// TIA Portal V19 export
FUNCTION_BLOCK "TYPIC_C904_BF_SPI"   // FB44, FBD
TITLE = TYPIC_C904_BF_SPI: Schoonvloeistofpompinstallatie
{ S7_Optimized_Access := 'TRUE' }
AUTHOR : OCOTECH
FAMILY : Typical
NAME : C904.801
// Logisch Object Besturing: C904.801
// 
// 								Het doel van de BF SPI (schoonvloeistofpompinstallatie) is om de
// 								algemene sturing te voorzien van de schoonvloeistofpompinstallatie.
// 								De algemene sturing omvat het weergeven van de algemene toestand en
// 								het aano en afschakelen van pompen in functie van het vloeistofpeil
// 								en het actieve regime.
// stored: MemoryReserve 10, SetENOAutomatically false
   VAR_INPUT
      CFG_TST_UTYD { ExternalAccessible := 'False'; ExternalVisible := 'False'; ExternalWritable := 'False'} : Time;   // Time-out standverandering pompinstallatie (transitiestatus onbereikt)
      CFG_TST_OK_TYD { ExternalAccessible := 'False'; ExternalVisible := 'False'; ExternalWritable := 'False'} : Time;   // Stabilisatietijd voor de toestand OK (bereikt)
      CFG_NIV_H { ExternalAccessible := 'False'; ExternalVisible := 'False'; ExternalWritable := 'False'} : Real;   // Grenswaarde voor dreigende overloop (minder dan 30m3 bergruimte)
      CFG_NIV_HH { ExternalAccessible := 'False'; ExternalVisible := 'False'; ExternalWritable := 'False'} : Real;   // Grenswaarde voor overloop
      CFG_NIV_ITYD { ExternalAccessible := 'False'; ExternalVisible := 'False'; ExternalWritable := 'False'} : Time;   // Inschakelvertraging storingen grenswaarde
      CFG_NIV_HYS { ExternalAccessible := 'False'; ExternalVisible := 'False'; ExternalWritable := 'False'} : Real;   // Hysteresis storingen grenswaarde
      CFG_DEB_H { ExternalAccessible := 'False'; ExternalVisible := 'False'; ExternalWritable := 'False'} : Real;   // Grenswaarde minimaal debiet bij 1 aangeschakelde pomp
      CFG_DEB_HH { ExternalAccessible := 'False'; ExternalVisible := 'False'; ExternalWritable := 'False'} : Real;   // Grenswaarde minimaal debiet bij meerdere aangeschakelde pompen
      CFG_ITYD_DEB { ExternalAccessible := 'False'; ExternalVisible := 'False'; ExternalWritable := 'False'} : Time;   // Tijdsvertraging voor alarm afvoer verstopt (pomp aangeschakeld en minimaal debiet niet bereikt)
      STU_CMD_AUT { ExternalAccessible := 'False'; ExternalVisible := 'False'; ExternalWritable := 'False'} : USInt;   // Groepscommando: schakel in automatisch
      STU_CMD_WRE { ExternalAccessible := 'False'; ExternalVisible := 'False'; ExternalWritable := 'False'} : USInt;   // Sturing regime
      STU_ALG_LCK_SIG { ExternalAccessible := 'False'; ExternalVisible := 'False'; ExternalWritable := 'False'} : USInt;   // Onderdruk alarmen
   END_VAR
   VAR_OUTPUT
      VAR_PWR { ExternalAccessible := 'False'; ExternalVisible := 'False'; ExternalWritable := 'False'} : Real;   // Som actuele vermogens van alle pompen
      STU_PMP1 { ExternalAccessible := 'False'; ExternalVisible := 'False'; ExternalWritable := 'False'} : USInt;   // Sturing pomp
      STU_PMP2 { ExternalAccessible := 'False'; ExternalVisible := 'False'; ExternalWritable := 'False'} : USInt;   // Sturing pomp
      STU_PMP3 { ExternalAccessible := 'False'; ExternalVisible := 'False'; ExternalWritable := 'False'} : USInt;   // Sturing pomp
      STU_IF_SPI { ExternalAccessible := 'False'; ExternalVisible := 'False'; ExternalWritable := 'False'} : USInt;   // Gewenst regime (naar interne sturing)
   END_VAR
   VAR_IN_OUT
      VAR_IF_SPI : "C904_VAR_IF_SPI_TYPIC";   // Struct met variabelen ontvangen van de interne sturing van de pompinstallatie
      VAR_PMP : Array[*] of "C904_VAR_PMP_TYPIC";   // Array met alle pompen, met alle variabelen van de pomp
      VAR_NIV : "C904_VAR_NIV_TYPIC";   // Struct met alle variabelen ontvangen van de subfunctie niveaumeting
      VAR_DEB : "C904_VAR_DEB_TYPIC";   // Struct met alle variabelen ontvangen van de subfunctie debietmeting
   END_VAR
   VAR
      BED : Struct   // Bedieningen
         ALG : Struct   // Gewenste stand
            X : "UDT_BED_ALG";
            KNOP { S7_SetPoint := 'True'} : Array[0..3] of "UDT_BED_KNOP";
         END_STRUCT;
      END_STRUCT;
      BED_ALG { ExternalWritable := 'False'} : "TYPIC_HF_BED_ALG_KNOP";   // Gewenste stand
      SIG { ExternalWritable := 'False'} : Struct   // Signaleringen
         AA01 : Bool;   // Gewenste stand niet bereikt (transitiestatus = niet bereikt)
         AA02 : Bool;   // Schoonvloeistofpompinstallatie dreigt over te lopen
         AA03 : Bool;   // Overschrijding capaciteit schoonvloeistofpompinstallatie (overloop)
         AA04 : Bool;   // Afvoer verstopt en dreiging overloop van de schoonvloeistofpompinstallatie
         AA05 : Bool;   // Afvoer verstopt
         AB01 : Bool;   // Schoonvloeistofpompinstallatie niet beschikbaar
         AB02 : Bool;   // Schoonvloeistofpompinstallatie beperkt beschikbaar
         A001 : Bool;   // Beveiliging aangesproken
         A002 : Bool;   // Beveiliging No-Break aangesproken
         A003 : Bool;   // Overspanningsbeveiliging aangesproken
         A004 : Bool;   // Schuif ALSB uitgeschakeld
         A005 : Bool;   // Schuif ALSB in test
         A006 : Bool;   // Schuif ALSB uitgereden
         A007 : Bool;   // Nisdeur niet gesloten
         A008 : Bool;   // Storing tracing
      END_STRUCT;
      VAR { ExternalWritable := 'False'} : Struct   // Variabelen
         BSC : USInt;   // Geeft de beschikbaarheid aan van het deelsysteem
         TST_BWA : USInt;   // De status van de transitie van het deelsysteem
         BMO : USInt;   // Bedieningsmode
         WRE_BWA : USInt;   // Actueel regime
         CAPA : USInt;   // Beschikbare pompcapaciteit
         STS_TRA : USInt;   // Status van de tracing
         STS_NIV : USInt;   // Vloeistofniveau bepaald door de stand van de vlotters
         WRE_SWA { ExternalAccessible := 'False'; ExternalVisible := 'False'} : USInt;   // Gewenst regime
         REQ_AAN { ExternalAccessible := 'False'; ExternalVisible := 'False'} : USInt;   // Gewenst aantal aangeschakelde pompen
         CAPA_OK { ExternalAccessible := 'False'; ExternalVisible := 'False'} : USInt;   // Aantal beschikbare pompen
         STS_AAN { ExternalAccessible := 'False'; ExternalVisible := 'False'} : USInt;   // Actueel aantal aangeschakelde pompen
      END_STRUCT;
      HF_TST { ExternalAccessible := 'False'; ExternalVisible := 'False'; ExternalWritable := 'False'} : "TYPIC_HF_TST";   // Hulpfunctie transitiestatus
   END_VAR
   // // BED.ALG.KNOP[0] : Auto
   // // BED.ALG.KNOP[1] : Leeghouden
   // // BED.ALG.KNOP[2] : Bergen
   // // BED.ALG.KNOP[3] : Uit
BEGIN

REGION Network 1: START
END_REGION

REGION Network 2: +++ Bedieningen +++
   // Vrijgave en verwerking van de bedieningen (centrale en
   // 										lokale bediening). De bedienwaardes worden daarna in de
   // 										verdere deelfunctionaliteiten gebruikt.
END_REGION

REGION Network 3: Knoppen BED_ALG(Gewenste stand)
   // Waardes en vrijge van de knoppen BED_ALG
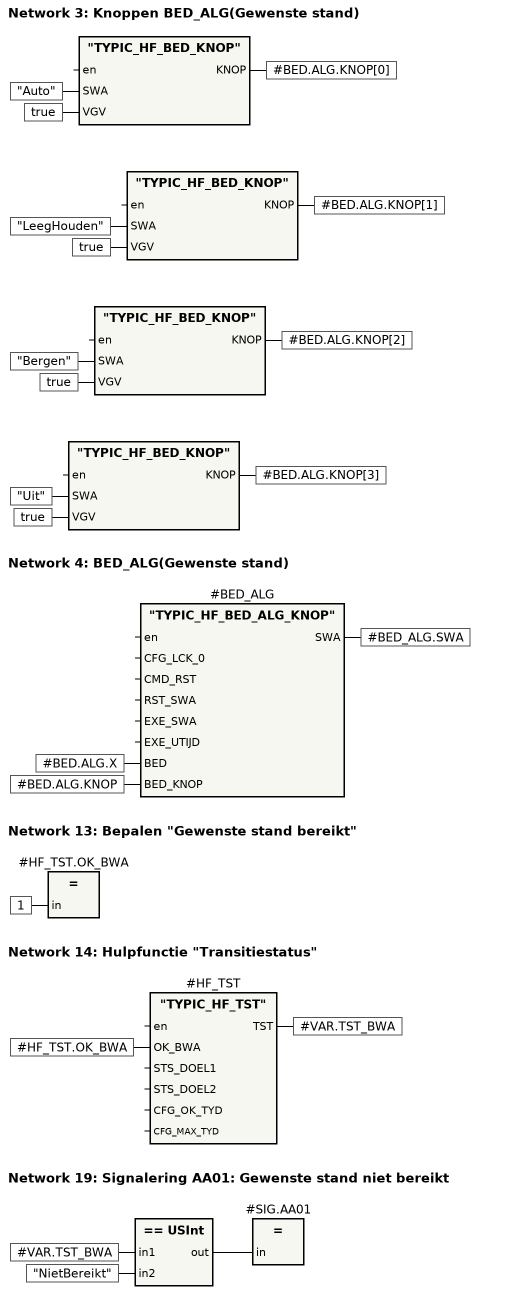
   "TYPIC_HF_BED_KNOP"(SWA := "Auto", VGV := true, KNOP => #BED.ALG.KNOP[0]);
   "TYPIC_HF_BED_KNOP"(SWA := "LeegHouden", VGV := true, KNOP => #BED.ALG.KNOP[1]);
   "TYPIC_HF_BED_KNOP"(SWA := "Bergen", VGV := true, KNOP => #BED.ALG.KNOP[2]);
   "TYPIC_HF_BED_KNOP"(SWA := "Uit", VGV := true, KNOP => #BED.ALG.KNOP[3]);
END_REGION

REGION Network 4: BED_ALG(Gewenste stand)
   // Verwerking BED_ALG
   #BED_ALG(BED := #BED.ALG.X, BED_KNOP := #BED.ALG.KNOP, SWA => #BED_ALG.SWA);   // "TYPIC_HF_BED_ALG_KNOP"
END_REGION

REGION Network 5: +++ Bepalen gewenst regime +++
   // Het gewenst regime (Leeghouden / Bergen / Uit)
END_REGION

REGION Network 6: +++ Bepalen actueel regime en bedieningsmode +++
   // Bepalen bedieningsmode (Automatisch / Manueel / Hand) en
   // 										daarna vastleggen van het actuele regime (Leeghouden /
   // 										Bergen / Uit).
END_REGION

REGION Network 7: +++ Berekeningen +++
   // Verscheidene berekeningen die nodig zijn voor de
   // 										functionele werking of info voor weergave via de centrale en
   // 										lokale bediening, zoals het aantal beschikbare pompen, het
   // 										actueel aantal aangeschakelde pompen en de beschikbare
   // 										pompcapaciteit.
END_REGION

REGION Network 8: +++ Bepalen vloeistofniveau +++
   // Het vloeistofniveau wordt bepaalt door, de status van de
   // 										verschillende vlotters (ontvangen via de niveaumeting) en de
   // 										vlotters droogloopbeveiliging van de pompen, om te zetten
   // 										naar een status.
END_REGION

REGION Network 9: +++ Pompsturing bij regime “Uit” +++
   // Alle pompen behorende tot de schoonvloeistofinstallatie
   // 										worden uitgeschakeld.
END_REGION

REGION Network 10: +++ Pompsturing bij regime “Bergen” +++
   // Pomp(en) aan- of uitschakelen op basis van de peilen LHW
   // 										en HHW van de niveaumeting.
END_REGION

REGION Network 11: +++ Pompsturing bij regime “Leeghouden” +++
   // Pomp(en) aan- of uitschakelen op basis van de peilen SW en
   // 										MSW en LHW van de niveaumeting.
END_REGION

REGION Network 12: +++ Bepalen transitiestatus +++
   // Transitiestatus (bereikt / niet bereikt / in transitie)
   // 										bepalen.
END_REGION

REGION Network 13: Bepalen "Gewenste stand bereikt"
   // Bepalen of de actuele stand in overeenstemming is met de
   // 										gewenste stand
   #HF_TST.OK_BWA := 1;
END_REGION

REGION Network 14: Hulpfunctie "Transitiestatus"
   // De transitiestatus geeft de relatie tussen een gewenste
   // 										stand (van een functionaliteit) en de actuele stand aan.
   #HF_TST(OK_BWA := #HF_TST.OK_BWA, TST => #VAR.TST_BWA);   // "TYPIC_HF_TST"
END_REGION

REGION Network 15: +++ Bepalen beschikbaarheidsstatus +++
   // Beschikbaarheidsstatus (beschikbaar / beperkt beschikbaar
   // 										/ niet beschikbaar) bepalen.
END_REGION

REGION Network 16 (SCL): Beschikbaarheidsstatus bepalen
   IF 
       //voorwaarden "Niet beschikbaar"
       TRUE
   THEN
       //Beschikbaarheidsstatus = Niet Beschikbaar
       #VAR.BSC:= "NietBeschikbaar";
   ELSIF
       //voorwaarden "Beperkt beschikbaar"
       TRUE
   THEN
       //Beschikbaarheidsstatus = Beperkt Beschikbaar
       #VAR.BSC:= "Beperkt";
   ELSE
       //Beschikbaarheidsstatus = Beschikbaar
       #VAR.BSC:= "Beschikbaar";
   END_IF;
END_REGION

REGION Network 17: +++ Signaleringen +++
   // Aanmaken signaleringen.
END_REGION

REGION Network 18 (SCL): Signaleringen voor de onderhoudsoperator
   // Signalering van de storingen ontvangen vanuit de interne
   // 										sturing
   #SIG.A001 := #VAR_IF_SPI.STO.A001;
   #SIG.A002 := #VAR_IF_SPI.STO.A002;
   #SIG.A003 := #VAR_IF_SPI.STO.A003;
   #SIG.A004 := #VAR_IF_SPI.STO.A004;
   #SIG.A005 := #VAR_IF_SPI.STO.A005;
   #SIG.A006 := #VAR_IF_SPI.STO.A006;
   #SIG.A007 := #VAR_IF_SPI.STO.A007;
   #SIG.A008 := #VAR_IF_SPI.STO.A008;
END_REGION

REGION Network 19: Signalering AA01: Gewenste stand niet bereikt
   #SIG.AA01 := #VAR.TST_BWA = "NietBereikt";
END_REGION

REGION Network 20: Signalering AB01 : Niet Beschikbaar
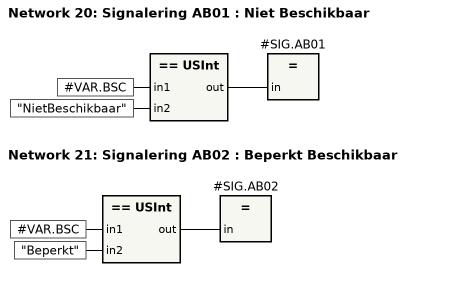
   #SIG.AB01 := #VAR.BSC = "NietBeschikbaar";
END_REGION

REGION Network 21: Signalering AB02 : Beperkt Beschikbaar
   #SIG.AB02 := #VAR.BSC = "Beperkt";
END_REGION

REGION Network 22: +++ Sturingen +++
   // Individuele commandos uitsturen naar iedere pomp om in- en
   // 										uit te schakelen.
END_REGION

REGION Network 23: EINDE
   // Variabelen van intern scada rakvlak naar outputs copieren
END_REGION
END_FUNCTION_BLOCK
